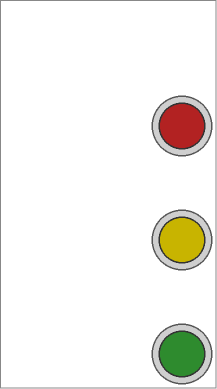
VISUALIZATION Visualization  // 217x389
    Lamp1 (147,91 70x70), variable: MAIN.Rosso, style: Lamp-Lamp1-Red
    Lamp1 (147,205 70x70), variable: MAIN.Giallo, style: Lamp-Lamp1-Yellow
    Lamp1 (147,319 70x70), variable: MAIN.Verde, style: Lamp-Lamp1-Green
END_VISUALIZATION

(* stored: Version 1.1.0.1, ProductVersion 3.1.4024.12
   Visu Visualization: Id {b4257c5b-f064-4636-a1b1-e6b6dc0e5152} *)
